// TIA Portal V20 export
TYPE "UDT_AxisPosition_OLD"
   STRUCT
      Axis_U : Struct
         PosExternalLoad : Real;
         PosExternalUnload : Real;
         PosSas : Real;
         PosBlowing : Real;
         PosControlUndrilled : Real;
         PosControlDrilled : Real;
         PosInternalLoadUndrilled : Real;
         PosInternalUnloadDrilled : Real;
         PosSemiAuto : Real;
         PosExtGateExt : Real;
         PosIntGateExt : Real;
         PosExtGateInt : Real;
         PosIntGateInt : Real;
      END_STRUCT;
      Axis_V : Struct
         PosShuttleUndrilled : Real;
         PosShuttleDrilled : Real;
         PosWashingVacuum : Real;
         PosWashingBrush : Real;
         PosHome : Real;
         PosChangeBackwall : Real;
      END_STRUCT;
      Axis_W : Struct
         PosUp : Real;
         PosShuttleUndrilled : Real;
         PosShuttleDrilled : Real;
         PosWashingVacuum : Real;
         PosWashingBrush : Real;
         PosChangeBackwall : Real;
      END_STRUCT;
      Axis_X : Struct
         PosChangeBackwall : Real;
      END_STRUCT;
      Axis_Y : Struct
         PosChangeBackwall : Real;
      END_STRUCT;
      Axis_ZM : Struct
         PosChangeBackwall : Real;
      END_STRUCT;
      Axis_ZL : Struct
         PosChangeBackwall : Real;
      END_STRUCT;
      Axis_B : Struct
         PosChangeBackwall : Real;
      END_STRUCT;
      Axis_C : Struct
         PosChangeBackwall : Real;
      END_STRUCT;
   END_STRUCT;
END_TYPE
